TYPE INTERNAL U_EcObject :
UNION
	iComponent	: I_Component;
	iEntity		: I_EntityNode;
END_UNION
END_TYPE

(* stored: Version 1.1.0.1
   DUT U_EcObject: Id {03758be6-2b89-43ee-b6ee-40fda7565e5b} *)
